// Mitsubishi GX Works2 project: 2023-06-27 #1 생산자동화기능사 9번   PLC: Q03UDV
// 생산자동화기능사

// global labels: Global1
VAR_GLOBAL
  PB1 AT X0 : BOOL;
  PB2 AT X1 : BOOL;
  정지 AT X2 : BOOL;
  공급후진 AT X3 : BOOL;
  공급전진 AT X4 : BOOL;
  가공후진 AT X5 : BOOL;
  가공전진 AT X6 : BOOL;
  송출후진 AT X7 : BOOL;
  송출전진 AT X8 : BOOL;
  배출후진 AT X9 : BOOL;
  배출전진 AT X0A : BOOL;
  매거진 AT X0B : BOOL;
  금속센서 AT X0F : BOOL;
  PB3 AT X10 : BOOL;
  적색 AT Y20 : BOOL;
  황색 AT Y21 : BOOL;
  녹색 AT Y22 : BOOL;
  공급1 AT Y23 : BOOL;
  공급2 AT Y24 : BOOL;
  가공 AT Y25 : BOOL;
  드릴 AT Y26 : BOOL;
  송출 AT Y27 : BOOL;
  배출 AT Y28 : BOOL;
  컨베이어 AT Y29 : BOOL;
END_VAR

PROGRAM 테스트동작
VAR
  PHASE : INT;
END_VAR
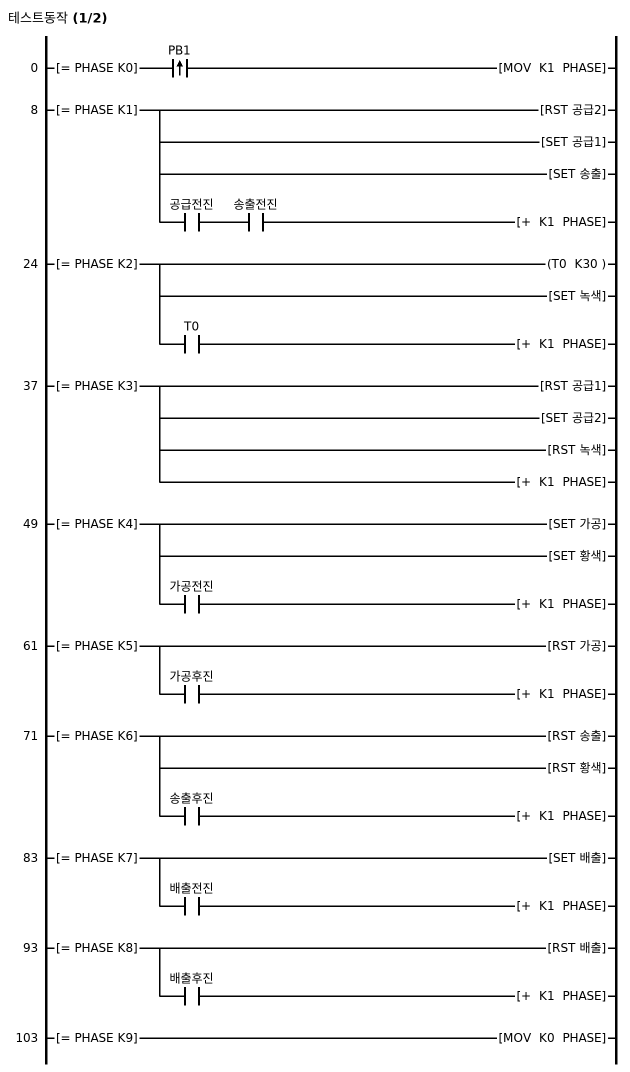
0     LD=     PHASE K0
      ANDP    PB1
      MOV     K1 PHASE
8     LD=     PHASE K1
      RST     공급2
      SET     공급1
      SET     송출
      AND     공급전진
      AND     송출전진
      +       K1 PHASE
24    LD=     PHASE K2
      OUT     T0 K30
      SET     녹색
      AND     T0
      +       K1 PHASE
37    LD=     PHASE K3
      RST     공급1
      SET     공급2
      RST     녹색
      +       K1 PHASE
49    LD=     PHASE K4
      SET     가공
      SET     황색
      AND     가공전진
      +       K1 PHASE
61    LD=     PHASE K5
      RST     가공
      AND     가공후진
      +       K1 PHASE
71    LD=     PHASE K6
      RST     송출
      RST     황색
      AND     송출후진
      +       K1 PHASE
83    LD=     PHASE K7
      SET     배출
      AND     배출전진
      +       K1 PHASE
93    LD=     PHASE K8
      RST     배출
      AND     배출후진
      +       K1 PHASE
103   LD=     PHASE K9
      MOV     K0 PHASE
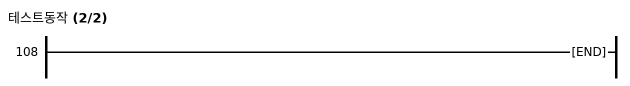
108   END
END_PROGRAM

PROGRAM 단속및연속동작
VAR
  PHASE : INT;
  MODE : INT;
END_VAR
VAR CONSTANT
  단속 : INT;
  연속 : INT := 1;
END_VAR
VAR
  LOOP : ARRAY [0..0] OF INT;
  BLINK : ARRAY [0..3] OF BOOL;
  PHASE1 : INT;
  드릴1 : BOOL;
END_VAR
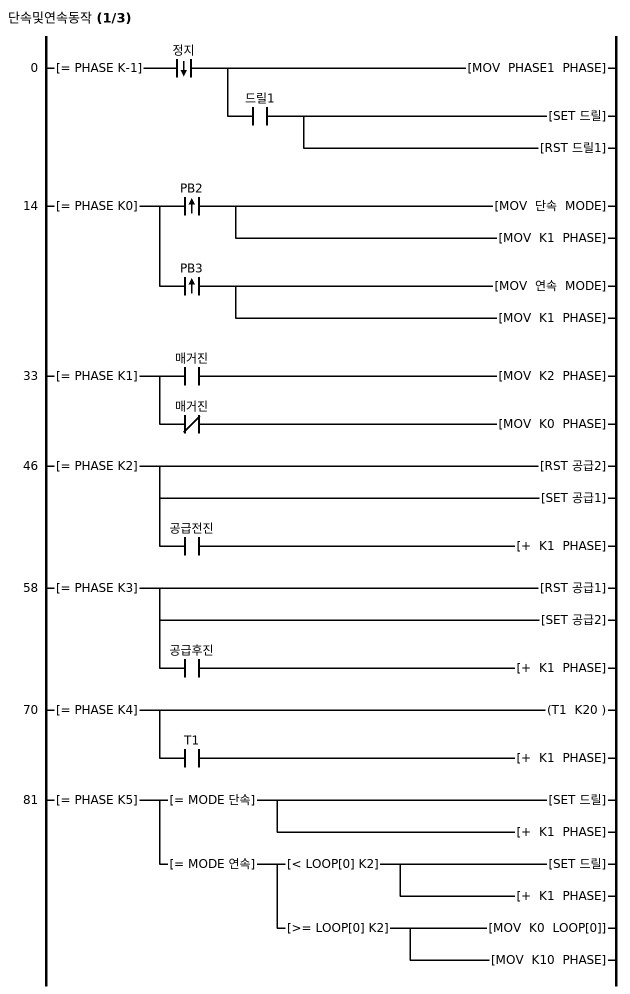
0     LD=     PHASE K-1
      ANDF    정지
      MOV     PHASE1 PHASE
      AND     드릴1
      SET     드릴
      RST     드릴1
14    LD=     PHASE K0
      MPS
      ANDP    PB2
      MOV     단속 MODE
      MOV     K1 PHASE
      MPP
      ANDP    PB3
      MOV     연속 MODE
      MOV     K1 PHASE
33    LD=     PHASE K1
      MPS
      AND     매거진
      MOV     K2 PHASE
      MPP
      ANI     매거진
      MOV     K0 PHASE
46    LD=     PHASE K2
      RST     공급2
      SET     공급1
      AND     공급전진
      +       K1 PHASE
58    LD=     PHASE K3
      RST     공급1
      SET     공급2
      AND     공급후진
      +       K1 PHASE
70    LD=     PHASE K4
      OUT     T1 K20
      AND     T1
      +       K1 PHASE
81    LD=     PHASE K5
      MPS
      AND=    MODE 단속
      SET     드릴
      +       K1 PHASE
      MPP
      AND=    MODE 연속
      MPS
      AND<    LOOP[0] K2
      SET     드릴
      +       K1 PHASE
      MPP
      AND>=   LOOP[0] K2
      MOV     K0 LOOP[0]
      MOV     K10 PHASE
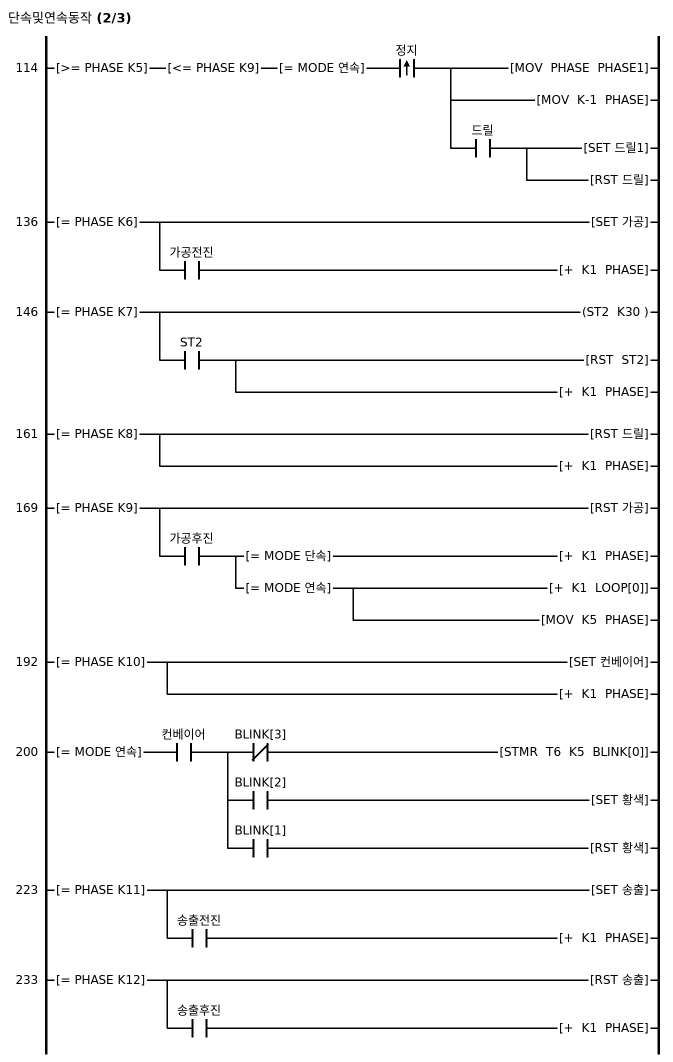
114   LD>=    PHASE K5
      AND<=   PHASE K9
      AND=    MODE 연속
      ANDP    정지
      MOV     PHASE PHASE1
      MOV     K-1 PHASE
      AND     드릴
      SET     드릴1
      RST     드릴
136   LD=     PHASE K6
      SET     가공
      AND     가공전진
      +       K1 PHASE
146   LD=     PHASE K7
      OUT     ST2 K30
      AND     ST2
      RST     ST2
      +       K1 PHASE
161   LD=     PHASE K8
      RST     드릴
      +       K1 PHASE
169   LD=     PHASE K9
      RST     가공
      AND     가공후진
      MPS
      AND=    MODE 단속
      +       K1 PHASE
      MPP
      AND=    MODE 연속
      +       K1 LOOP[0]
      MOV     K5 PHASE
192   LD=     PHASE K10
      SET     컨베이어
      +       K1 PHASE
200   LD=     MODE 연속
      AND     컨베이어
      MPS
      ANI     BLINK[3]
      STMR    T6 K5 BLINK[0]
      MRD
      AND     BLINK[2]
      SET     황색
      MPP
      AND     BLINK[1]
      RST     황색
223   LD=     PHASE K11
      SET     송출
      AND     송출전진
      +       K1 PHASE
233   LD=     PHASE K12
      RST     송출
      AND     송출후진
      +       K1 PHASE
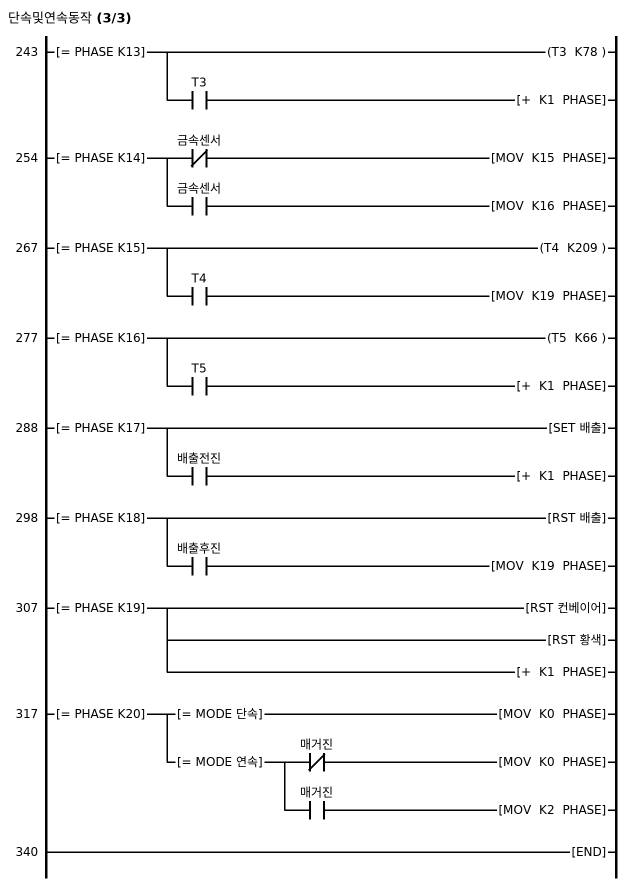
243   LD=     PHASE K13
      OUT     T3 K78
      AND     T3
      +       K1 PHASE
254   LD=     PHASE K14
      MPS
      ANI     금속센서
      MOV     K15 PHASE
      MPP
      AND     금속센서
      MOV     K16 PHASE
267   LD=     PHASE K15
      OUT     T4 K209
      AND     T4
      MOV     K19 PHASE
277   LD=     PHASE K16
      OUT     T5 K66
      AND     T5
      +       K1 PHASE
288   LD=     PHASE K17
      SET     배출
      AND     배출전진
      +       K1 PHASE
298   LD=     PHASE K18
      RST     배출
      AND     배출후진
      MOV     K19 PHASE
307   LD=     PHASE K19
      RST     컨베이어
      RST     황색
      +       K1 PHASE
317   LD=     PHASE K20
      MPS
      AND=    MODE 단속
      MOV     K0 PHASE
      MPP
      AND=    MODE 연속
      MPS
      ANI     매거진
      MOV     K0 PHASE
      MPP
      AND     매거진
      MOV     K2 PHASE
340   END
END_PROGRAM
